FUNCTION CASIN : complex
VAR_INPUT
	X : complex;
END_VAR
VAR
	Y : complex;
END_VAR

(*
version 1.0	21 feb 2008
programmer 	hugo
tested by	oscat

this function calculates the arcus sinus function of a complex number

*)

y.re := -x.im;
y.im := x.re;
y := CASINH(y);
CASIN.re := y.im;
CASIN.im := -y.re;



(* revision history
hm	21. feb 2008	rev 1.0
	original version


*)

END_FUNCTION

(* stored: Version 1.1.0.1, ProductVersion 3.1.4022.7
   POU CASIN: Id {288383d2-f5e5-4859-b8d9-1f7bdf4a62e8}, SpecialFunc None *)
